# EPICS substitutions: fastFeedbackApp/Db/common/fbckSettledSumInj.substitutions
file fbckSettledInjStatus.template {
        pattern { LOOP, INJ}
                { $(LP), "FBCK:IN20:TR01:CVGCALC"}
}
